(* IEC 61131-3 sources: cc_kush_rewrite/POUs/Bunker/POU/Hardware, 4 files *)

(* ---- FB_BunkerMotorErrors.st ---- *)
FUNCTION_BLOCK FB_BunkerMotorErrors
VAR_INPUT
	Bunker : REFERENCE TO ST_Bunker;
	xReset : BOOL; // Команда сброса зафиксированных ошибок
END_VAR
VAR_OUTPUT
	// Ошибки вибропитателей (индивидуально)
	xErrorVibFeeder1 : BOOL;
	xErrorVibFeeder2 : BOOL;
	xErrorMotorVibFeeder_Any : BOOL; // Ошибка хотя бы одного вибропитателя

	// Ошибки вибраторов (индивидуально)
	xErrorVibrator1 : BOOL;
	xErrorVibrator2 : BOOL;
	xErrorVibrator3 : BOOL;
	xErrorVibrator4 : BOOL;
	xErrorMotorVibrator_Any : BOOL; // Ошибка хотя бы одного вибратора

	// Ошибки бункера
	xErrorBunker : BOOL; // Ошибка бункера (люк, вес)

	// Состояние автоматических выключателей (QF)
	xQF_OkVibFeeder1 : BOOL;
	xQF_OkVibFeeder2 : BOOL;
	xQF_OkVibFeeder_All : BOOL;

	xQF_OkVibrator1 : BOOL;
	xQF_OkVibrator2 : BOOL;
	xQF_OkVibrator3 : BOOL;
	xQF_OkVibrator4 : BOOL;
	xQF_OkVibrator_All : BOOL;

	xQF_Ok_All : BOOL; // Все QF включены

	// Готовность VFD
	xVFD_ReadyVibFeeder1 : BOOL;
	xVFD_ReadyVibFeeder2 : BOOL;
	xVFD_ReadyVibFeeder_All : BOOL;

	xVFD_ReadyVibrator1 : BOOL;
	xVFD_ReadyVibrator2 : BOOL;
	xVFD_ReadyVibrator3 : BOOL;
	xVFD_ReadyVibrator4 : BOOL;
	xVFD_ReadyVibrator_All : BOOL;

	xVFD_Ready_All : BOOL; // Все VFD готовы
END_VAR
VAR
	// Внутренние переменные для текущих состояний ошибок (без фиксации)
	_xCurrentErrorVibFeeder1 : BOOL;
	_xCurrentErrorVibFeeder2 : BOOL;
	_xCurrentErrorVibrator1 : BOOL;
	_xCurrentErrorVibrator2 : BOOL;
	_xCurrentErrorVibrator3 : BOOL;
	_xCurrentErrorVibrator4 : BOOL;
	_xCurrentErrorBunker : BOOL;

	// RS-триггеры для фиксации ошибок
	_fbLatchErrorVibFeeder1 : RS;
	_fbLatchErrorVibFeeder2 : RS;
	_fbLatchErrorVibrator1 : RS;
	_fbLatchErrorVibrator2 : RS;
	_fbLatchErrorVibrator3 : RS;
	_fbLatchErrorVibrator4 : RS;
	_fbLatchErrorBunker : RS;
END_VAR

// ========================================
// FB_BunkerMotorErrors - Проверка ошибок моторов бункера
// ========================================
//
// НАЗНАЧЕНИЕ:
// - Проверка всех моторов бункера на ошибки
// - Фиксация ошибок через RS-триггеры (память до сброса)
// - Формирование индивидуальных флагов ошибок
// - Агрегирование ошибок
//
// МОТОРЫ:
// - MotorVibFeeder[1..2]: Вибропитатели (7.5 кВт)
// - MotorVibrator[1..4]: Вибраторы (0.62 кВт)
//
// ПРОВЕРЯЕМЫЕ ОШИБКИ:
// - Ошибка VFD (fbStateFailure: NC контакт - 0 = ошибка, 1 = норма)
// - Локальная ошибка VFD (xStateFailureLocal: программная установка ошибки)
//
// ЛОГИКА ФИКСАЦИИ:
// - При возникновении ошибки она фиксируется (SET в RS-триггер)
// - Ошибка сохраняется даже после устранения неисправности
// - Сброс всех зафиксированных ошибок через вход xReset
//
// ========================================

// ========================================
// ПРОВЕРКА ОШИБОК ВИБРОПИТАТЕЛЕЙ
// ========================================

// Вибропитатель 1
// fbStateFailure - NC контакт: 0 = ошибка VFD, 1 = норма
// Используем инвертированный сигнал (qxInvertedSignal: TRUE = ошибка)
_xCurrentErrorVibFeeder1 := Bunker.MotorVibFeeder[1].VFD.fbStateFailure.qxInvertedSignal
                         OR Bunker.MotorVibFeeder[1].VFD.xStateFailureLocal;

// Вибропитатель 2
_xCurrentErrorVibFeeder2 := Bunker.MotorVibFeeder[2].VFD.fbStateFailure.qxInvertedSignal
                         OR Bunker.MotorVibFeeder[2].VFD.xStateFailureLocal;

// Фиксируем ошибки через RS-триггеры
_fbLatchErrorVibFeeder1(SET := _xCurrentErrorVibFeeder1, RESET1 := xReset);
_fbLatchErrorVibFeeder2(SET := _xCurrentErrorVibFeeder2, RESET1 := xReset);

// Выходы - зафиксированные ошибки
xErrorVibFeeder1 := _fbLatchErrorVibFeeder1.Q1;
xErrorVibFeeder2 := _fbLatchErrorVibFeeder2.Q1;

xErrorMotorVibFeeder_Any := xErrorVibFeeder1 OR xErrorVibFeeder2;

// ========================================
// ПРОВЕРКА ОШИБОК ВИБРАТОРОВ
// ========================================

// Вибратор 1
_xCurrentErrorVibrator1 := Bunker.MotorVibrator[1].VFD.fbStateFailure.qxInvertedSignal
                        OR Bunker.MotorVibrator[1].VFD.xStateFailureLocal;

// Вибратор 2
_xCurrentErrorVibrator2 := Bunker.MotorVibrator[2].VFD.fbStateFailure.qxInvertedSignal
                        OR Bunker.MotorVibrator[2].VFD.xStateFailureLocal;

// Вибратор 3
_xCurrentErrorVibrator3 := Bunker.MotorVibrator[3].VFD.fbStateFailure.qxInvertedSignal
                        OR Bunker.MotorVibrator[3].VFD.xStateFailureLocal;

// Вибратор 4
_xCurrentErrorVibrator4 := Bunker.MotorVibrator[4].VFD.fbStateFailure.qxInvertedSignal
                        OR Bunker.MotorVibrator[4].VFD.xStateFailureLocal;

// Фиксируем ошибки через RS-триггеры
_fbLatchErrorVibrator1(SET := _xCurrentErrorVibrator1, RESET1 := xReset);
_fbLatchErrorVibrator2(SET := _xCurrentErrorVibrator2, RESET1 := xReset);
_fbLatchErrorVibrator3(SET := _xCurrentErrorVibrator3, RESET1 := xReset);
_fbLatchErrorVibrator4(SET := _xCurrentErrorVibrator4, RESET1 := xReset);

// Выходы - зафиксированные ошибки
xErrorVibrator1 := _fbLatchErrorVibrator1.Q1;
xErrorVibrator2 := _fbLatchErrorVibrator2.Q1;
xErrorVibrator3 := _fbLatchErrorVibrator3.Q1;
xErrorVibrator4 := _fbLatchErrorVibrator4.Q1;

xErrorMotorVibrator_Any := xErrorVibrator1 OR xErrorVibrator2 OR xErrorVibrator3 OR xErrorVibrator4;

// ========================================
// ПРОВЕРКА ОШИБОК БУНКЕРА
// ========================================

// Проверка положения люка (1 = закрыт, 0 = открыт)
// Открытый люк = ошибка
_xCurrentErrorBunker := NOT Bunker.fbStateHatch.qxSignal;

// Фиксируем ошибку через RS-триггер
_fbLatchErrorBunker(SET := _xCurrentErrorBunker, RESET1 := xReset);

// Выход - зафиксированная ошибка
xErrorBunker := _fbLatchErrorBunker.Q1;

// ========================================
// ПРОВЕРКА ГОТОВНОСТИ VFD
// ========================================
// fbStateRdyToStart - NO контакт: 1 = готов к пуску, 0 = не готов
// Готовность проверяется в реальном времени (без фиксации)

// Готовность VFD вибропитателей
xVFD_ReadyVibFeeder1 := Bunker.MotorVibFeeder[1].VFD.fbStateRdyToStart.qxSignal;
xVFD_ReadyVibFeeder2 := Bunker.MotorVibFeeder[2].VFD.fbStateRdyToStart.qxSignal;
xVFD_ReadyVibFeeder_All := xVFD_ReadyVibFeeder1 AND xVFD_ReadyVibFeeder2;

// Готовность VFD вибраторов
xVFD_ReadyVibrator1 := Bunker.MotorVibrator[1].VFD.fbStateRdyToStart.qxSignal;
xVFD_ReadyVibrator2 := Bunker.MotorVibrator[2].VFD.fbStateRdyToStart.qxSignal;
xVFD_ReadyVibrator3 := Bunker.MotorVibrator[3].VFD.fbStateRdyToStart.qxSignal;
xVFD_ReadyVibrator4 := Bunker.MotorVibrator[4].VFD.fbStateRdyToStart.qxSignal;
xVFD_ReadyVibrator_All := xVFD_ReadyVibrator1 AND xVFD_ReadyVibrator2 AND xVFD_ReadyVibrator3 AND xVFD_ReadyVibrator4;

// Общая готовность всех VFD
xVFD_Ready_All := xVFD_ReadyVibFeeder_All AND xVFD_ReadyVibrator_All;

// ========================================
// ПРОВЕРКА СОСТОЯНИЯ АВТОМАТИЧЕСКИХ ВЫКЛЮЧАТЕЛЕЙ (QF)
// ========================================
// fbStateQF - NO контакт: 1 = QF включен, 0 = QF выключен
// Состояние проверяется в реальном времени (без фиксации)
// Выключенный QF - не ошибка, но запуск мотора невозможен

// Состояние QF вибропитателей
xQF_OkVibFeeder1 := Bunker.MotorVibFeeder[1].fbStateQF.qxSignal;
xQF_OkVibFeeder2 := Bunker.MotorVibFeeder[2].fbStateQF.qxSignal;
xQF_OkVibFeeder_All := xQF_OkVibFeeder1 AND xQF_OkVibFeeder2;

// Состояние QF вибраторов
xQF_OkVibrator1 := Bunker.MotorVibrator[1].fbStateQF.qxSignal;
xQF_OkVibrator2 := Bunker.MotorVibrator[2].fbStateQF.qxSignal;
xQF_OkVibrator3 := Bunker.MotorVibrator[3].fbStateQF.qxSignal;
xQF_OkVibrator4 := Bunker.MotorVibrator[4].fbStateQF.qxSignal;
xQF_OkVibrator_All := xQF_OkVibrator1 AND xQF_OkVibrator2 AND xQF_OkVibrator3 AND xQF_OkVibrator4;

// Общее состояние всех QF
xQF_Ok_All := xQF_OkVibFeeder_All AND xQF_OkVibrator_All;

END_FUNCTION_BLOCK

(* ---- FB_BunkerSensors.st ---- *)
FUNCTION_BLOCK FB_BunkerSensors
VAR_INPUT
	Bunker : REFERENCE TO ST_Bunker;
	xReset : BOOL;
END_VAR
VAR_OUTPUT
	xErrorHatch : BOOL;     // Ошибка положения люка
END_VAR

// ========================================
// FB_BunkerSensors - Обработка датчиков безопасности бункера
// ========================================
//
// НАЗНАЧЕНИЕ:
// - Обработка датчиков безопасности (люк)
// - Аналог FB_DumperSensors / FB_ConveyorSensors
// - Предоставляет единую точку для проверки датчиков
//
// ВХОДЫ:
// - Bunker: ссылка на структуру бункера
// - xReset: команда сброса ошибок
//
// ВЫХОДЫ:
// - xErrorHatch: ошибка положения люка
//
// ========================================

// ========================================
// ПРОВЕРКА ПОЛОЖЕНИЯ ЛЮКА
// ========================================

// Проверка положения люка (1 = закрыт, 0 = открыт)
// Если люк открыт - ошибка
xErrorHatch := NOT Bunker.fbStateHatch.qxSignal;

// ПРИМЕЧАНИЕ: В будущем здесь могут быть добавлены другие датчики безопасности

END_FUNCTION_BLOCK

(* ---- FB_BunkerVibFeederMotors.st ---- *)
FUNCTION_BLOCK FB_BunkerVibFeederMotors
VAR_INPUT
	Bunker : REFERENCE TO ST_Bunker;
	xStart : BOOL;              // Команда запуска
	xStop : BOOL;               // Команда остановки
	xEmergencyStop : BOOL;      // Аварийная остановка
	xReset : BOOL;              // Сброс ошибок
	rTargetFrequency : REAL;    // Целевая частота (Гц)
END_VAR
VAR_OUTPUT
	eStage : E_StageActuator;   // IDLE/STARTING/WORK/STOPPING/FAULT
	rCurrentFrequency : REAL;   // Средняя частота двух моторов
	xStartingTimeout : BOOL;    // Флаг тайм-аута запуска
	xStoppingTimeout : BOOL;    // Флаг тайм-аута остановки
END_VAR
VAR
	STAGE : E_StageActuator := E_StageActuator.IDLE;

	// Таймеры контроля времени запуска/остановки
	tonTimerStarting : TON;     // Контроль времени запуска (STARTING → WORK)
	tonTimerStopping : TON;     // Контроль времени остановки (STOPPING → IDLE)
END_VAR

// ========================================
// FB_BunkerVibFeederMotors - Управление моторами вибропитателей бункера
// ========================================
//
// НАЗНАЧЕНИЕ:
// - Управление двумя вибропитателями (7.5 кВт каждый)
// - Прямой пуск/остановка (без плавного разгона)
// - Не знает про ППЗ и верхнеуровневую логику
// - Просто выполняет команды START/STOP
//
// ВХОДЫ:
// - xStart: команда запуска моторов
// - xStop: команда остановки моторов
// - xEmergencyStop: аварийная остановка
// - xReset: сброс аварии
// - rTargetFrequency: целевая частота (Гц)
//
// ВЫХОДЫ:
// - eStage: текущая стадия (IDLE/STARTING/WORK/STOPPING/FAULT)
// - rCurrentFrequency: текущая частота моторов (среднее)
// - xStartingTimeout: флаг тайм-аута запуска
// - xStoppingTimeout: флаг тайм-аута остановки
//
// ========================================

// ========================================
// ПРИОРИТЕТНАЯ ОБРАБОТКА АВАРИЙНОЙ ОСТАНОВКИ
// ========================================

IF xEmergencyStop THEN
	// Аварийная остановка: немедленное выключение VFD
	Bunker.MotorVibFeeder[1].VFD.qxStart := FALSE;
	Bunker.MotorVibFeeder[2].VFD.qxStart := FALSE;

	// Переход в FAULT
	STAGE := E_StageActuator.FAULT;
	tonTimerStarting(IN := FALSE);
	tonTimerStopping(IN := FALSE);
END_IF

// ========================================
// ПРОВЕРКА ТАЙМ-АУТОВ ВЫПОЛНЕНИЯ КОМАНД
// ========================================

// Тайм-аут запуска: если слишком долго в STARTING → аварийная остановка
tonTimerStarting(
	IN := (STAGE = E_StageActuator.STARTING),
	PT := TIME_TIMEOUT_START_BUNKER
);

IF tonTimerStarting.Q THEN
	xStartingTimeout := TRUE;
	// Аварийная остановка: немедленное выключение VFD
	Bunker.MotorVibFeeder[1].VFD.qxStart := FALSE;
	Bunker.MotorVibFeeder[2].VFD.qxStart := FALSE;
	// Переход в FAULT
	STAGE := E_StageActuator.FAULT;
	tonTimerStarting(IN := FALSE);
END_IF

// Тайм-аут остановки: если слишком долго в STOPPING → аварийная остановка
tonTimerStopping(
	IN := (STAGE = E_StageActuator.STOPPING),
	PT := TIME_TIMEOUT_STOP_BUNKER
);

IF tonTimerStopping.Q THEN
	xStoppingTimeout := TRUE;
	// Аварийная остановка: немедленное выключение VFD
	Bunker.MotorVibFeeder[1].VFD.qxStart := FALSE;
	Bunker.MotorVibFeeder[2].VFD.qxStart := FALSE;
	// Переход в FAULT
	STAGE := E_StageActuator.FAULT;
	tonTimerStopping(IN := FALSE);
END_IF

// ========================================
// АВТОМАТ УПРАВЛЕНИЯ МОТОРАМИ
// ========================================

CASE STAGE OF
	E_StageActuator.IDLE:
		// Сброс команд
		Bunker.MotorVibFeeder[1].VFD.qxStart := FALSE;
		Bunker.MotorVibFeeder[2].VFD.qxStart := FALSE;

		// Команда запуска
		IF xStart AND NOT xEmergencyStop THEN
			STAGE := E_StageActuator.STARTING;
		END_IF

	E_StageActuator.STARTING:
		// Проверка команды остановки во время запуска
		IF xStop THEN
			// Прервать запуск и перейти к остановке
			STAGE := E_StageActuator.STOPPING;
		END_IF

		// Команда ПУСК на VFD
		Bunker.MotorVibFeeder[1].VFD.qxStart := TRUE;
		Bunker.MotorVibFeeder[2].VFD.qxStart := TRUE;

		// Проверка обратной связи VFD
		IF Bunker.MotorVibFeeder[1].VFD.fbStateIsWorking.qxSignal
		   AND Bunker.MotorVibFeeder[2].VFD.fbStateIsWorking.qxSignal
		THEN
			// Сброс таймера запуска (успешный запуск)
			tonTimerStarting(IN := FALSE);
			STAGE := E_StageActuator.WORK;
		END_IF

	E_StageActuator.WORK:
		// Нормальная работа
		// Команда остановки - переход в STOPPING
		IF xStop THEN
			STAGE := E_StageActuator.STOPPING;
		END_IF

	E_StageActuator.STOPPING:
		// Остановка VFD
		Bunker.MotorVibFeeder[1].VFD.qxStart := FALSE;
		Bunker.MotorVibFeeder[2].VFD.qxStart := FALSE;

		// Проверка остановки VFD (обратная связь)
		IF NOT Bunker.MotorVibFeeder[1].VFD.fbStateIsWorking.qxSignal
		   AND NOT Bunker.MotorVibFeeder[2].VFD.fbStateIsWorking.qxSignal
		THEN
			// Сброс таймера остановки (успешная остановка)
			tonTimerStopping(IN := FALSE);
			STAGE := E_StageActuator.IDLE;
		END_IF

	E_StageActuator.FAULT:
		// Состояние аварии - ожидание сброса
		// Выход из FAULT по команде xReset
		IF xReset THEN
			STAGE := E_StageActuator.IDLE;
			xStartingTimeout := FALSE; // Сброс флага тайм-аута запуска
			xStoppingTimeout := FALSE; // Сброс флага тайм-аута остановки
		END_IF
END_CASE;

// ========================================
// ЗАДАНИЕ ЧАСТОТЫ МОТОРОВ
// ========================================

// Установка частоты напрямую (без плавного разгона)
// В режимах STARTING и WORK частота = rTargetFrequency
// В остальных режимах (IDLE, STOPPING, FAULT) частота = 0
IF STAGE = E_StageActuator.STARTING OR STAGE = E_StageActuator.WORK THEN
	Bunker.MotorVibFeeder[1].VFD.qrOutFrequency := rTargetFrequency;
	Bunker.MotorVibFeeder[2].VFD.qrOutFrequency := rTargetFrequency;
ELSE
	Bunker.MotorVibFeeder[1].VFD.qrOutFrequency := 0.0;
	Bunker.MotorVibFeeder[2].VFD.qrOutFrequency := 0.0;
END_IF;

// ========================================
// ВЫХОДЫ
// ========================================

// Текущая стадия
eStage := STAGE;

// Текущая частота (среднее значение двух моторов)
rCurrentFrequency := (Bunker.MotorVibFeeder[1].VFD.rActualFrequency
                    + Bunker.MotorVibFeeder[2].VFD.rActualFrequency) / 2.0;

END_FUNCTION_BLOCK

(* ---- FB_BunkerVibratorMotors.st ---- *)
FUNCTION_BLOCK FB_BunkerVibratorMotors
VAR_INPUT
	Bunker : REFERENCE TO ST_Bunker;
	xEmergencyStop : BOOL;              // Аварийная остановка
	xReset : BOOL;                      // Сброс ошибок
	eVibratorMode : E_StateRemote;      // Auto/Manual/Repair
	xManualStart : BOOL;                // СТАРТ в ручном режиме
	xManualStop : BOOL;                 // СТОП в ручном режиме
	xSelectedVibrators : ARRAY[1..4] OF BOOL;  // Выбор вибраторов (галочки)
	rTargetFrequency : REAL;            // Целевая частота
	stVibratorSettings : ST_BunkerVibratorSettings; // Параметры цикла
	xEnableAutoMode : BOOL;             // Разрешение автоматического режима (только в WORK вибропитателей)
END_VAR
VAR_OUTPUT
	eStage : E_StageActuator;           // IDLE/STARTING/WORK/STOPPING/FAULT
	xVibratorAutoActive : BOOL;         // Флаг активной работы (Auto)
	xVibratorManualRunActive : BOOL;    // Флаг активной работы (Manual)
END_VAR
VAR
	STAGE : E_StageActuator := E_StageActuator.IDLE;  // Текущая стадия
	tonVibratorActive : TON;            // Таймер активной работы (Auto)
	tonVibratorPause : TON;             // Таймер паузы (Auto)
	i : INT;

	// Переменные для последовательного запуска вибраторов
	tonSequentialStart : TON;           // Таймер шага последовательного запуска
	nSequentialIndex : INT := 0;        // Текущий индекс в последовательности запуска (0 = не запущен, 1-4 = номер вибратора)
	axVibratorStarted : ARRAY[1..4] OF BOOL; // Флаги запущенных вибраторов в текущем цикле ACTIVE
	xSequentialStartComplete : BOOL;    // Все выбранные вибраторы запущены
END_VAR

// ========================================
// FB_BunkerVibratorMotors - Управление вибраторами бункера
// ========================================
//
// НАЗНАЧЕНИЕ:
// - Управление 4 вибраторами (0.62 кВт каждый)
// - 3 режима: Auto (цикл), Manual (выборочное управление), Repair (остановка)
// - Auto режим: ACTIVE (работа) ↔ PAUSE (пауза) циклически
// - Manual режим: индивидуальный выбор через галочки + СТАРТ/СТОП
// - Не знает про вибропитатели и верхнеуровневую логику
//
// ВХОДЫ:
// - xEmergencyStop: аварийная остановка
// - xReset: сброс ошибок
// - eVibratorMode: режим управления (Auto/Manual/Repair)
// - xManualStart: команда СТАРТ в ручном режиме
// - xManualStop: команда СТОП в ручном режиме
// - xSelectedVibrators[1..4]: выбор вибраторов (галочки)
// - rTargetFrequency: целевая частота (Гц)
// - stVibratorSettings: параметры цикла (TIME_ACTIVE, TIME_PAUSE_VIBRATOR и т.д.)
// - xEnableAutoMode: разрешение автоматического режима (TRUE только в WORK вибропитателей)
//
// ВЫХОДЫ:
// - eStage: текущая стадия (IDLE/STARTING/WORK/STOPPING/FAULT)
// - xVibratorAutoActive: флаг активной работы в авто режиме
// - xVibratorManualRunActive: флаг активной работы в ручном режиме
//
// ========================================

// ========================================
// ПРИОРИТЕТНАЯ ОБРАБОТКА АВАРИЙНОЙ ОСТАНОВКИ
// ========================================

IF xEmergencyStop THEN
	// Остановка всех VFD вибраторов
	Bunker.MotorVibrator[1].VFD.qxStart := FALSE;
	Bunker.MotorVibrator[2].VFD.qxStart := FALSE;
	Bunker.MotorVibrator[3].VFD.qxStart := FALSE;
	Bunker.MotorVibrator[4].VFD.qxStart := FALSE;

	// Сброс таймеров и флагов
	tonVibratorActive(IN := FALSE);
	tonVibratorPause(IN := FALSE);
	tonSequentialStart(IN := FALSE);
	xVibratorManualRunActive := FALSE;
	xVibratorAutoActive := FALSE;
	nSequentialIndex := 0;
	xSequentialStartComplete := FALSE;
	FOR i := 1 TO 4 BY 1 DO
		axVibratorStarted[i] := FALSE;
	END_FOR;

	// Переход в FAULT
	STAGE := E_StageActuator.FAULT;
END_IF

// ========================================
// НОРМАЛЬНАЯ РАБОТА ВИБРАТОРОВ
// ========================================

IF NOT xEmergencyStop THEN
	CASE eVibratorMode OF
		// ========================================
		// РЕЖИМ АВТОМАТИЧЕСКИЙ - циклическая работа по таймеру
		// ========================================
		E_StateRemote.Auto:
			// Автоматический режим работает только при разрешении (в WORK вибропитателей)
			IF xEnableAutoMode THEN
				// Установка частоты для вибраторов в автоматическом режиме
				FOR i := 1 TO AMOUNT_BUNKER_MOTOR_VIBRATOR BY 1 DO
					Bunker.MotorVibrator[i].VFD.qrOutFrequency := rTargetFrequency;
				END_FOR;

				// Таймеры автоматического цикла
				tonVibratorActive(PT := stVibratorSettings.TIME_ACTIVE);
				tonVibratorPause(PT := stVibratorSettings.TIME_PAUSE_VIBRATOR);
				tonSequentialStart(PT := TIME_VIBRATOR_SEQUENTIAL_START_STEP);

				// Логика автоматического цикла (ACTIVE ↔ PAUSE)
				IF NOT xVibratorAutoActive THEN
					// Состояние PAUSE - ждем окончания паузы
					IF tonVibratorPause.Q THEN
						// Пауза завершена - переход в ACTIVE
						tonVibratorPause(IN := FALSE);
						xVibratorAutoActive := TRUE;

						// Сброс состояния последовательного запуска
						nSequentialIndex := 0;
						xSequentialStartComplete := FALSE;
						FOR i := 1 TO 4 BY 1 DO
							axVibratorStarted[i] := FALSE;
						END_FOR;
						tonSequentialStart(IN := FALSE);
						tonVibratorActive(IN := FALSE); // Таймер ACTIVE запустится после завершения последовательного запуска

						// Переход в WORK (вибраторы будут запускаться последовательно)
						STAGE := E_StageActuator.WORK;
					ELSIF NOT tonVibratorPause.IN THEN
						// Первый запуск - сразу в ACTIVE
						xVibratorAutoActive := TRUE;

						// Сброс состояния последовательного запуска
						nSequentialIndex := 0;
						xSequentialStartComplete := FALSE;
						FOR i := 1 TO 4 BY 1 DO
							axVibratorStarted[i] := FALSE;
						END_FOR;
						tonSequentialStart(IN := FALSE);
						tonVibratorActive(IN := FALSE); // Таймер ACTIVE запустится после завершения последовательного запуска

						// Переход в WORK (вибраторы будут запускаться последовательно)
						STAGE := E_StageActuator.WORK;
					ELSE
						// Пауза активна - IDLE
						STAGE := E_StageActuator.IDLE;
					END_IF;
				ELSE
					// Состояние ACTIVE - последовательный запуск вибраторов

					// Логика последовательного запуска (если ещё не все запущены)
					IF NOT xSequentialStartComplete THEN
						// Проверка таймера для запуска следующего вибратора
						IF NOT tonSequentialStart.IN OR tonSequentialStart.Q THEN
							// Сброс таймера и поиск следующего выбранного вибратора
							tonSequentialStart(IN := FALSE);

							// Ищем следующий выбранный вибратор, который ещё не запущен
							FOR i := 1 TO 4 BY 1 DO
								IF xSelectedVibrators[i] AND NOT axVibratorStarted[i] THEN
									// Найден следующий вибратор для запуска
									Bunker.MotorVibrator[i].VFD.qxStart := TRUE;
									axVibratorStarted[i] := TRUE;
									nSequentialIndex := i;
									tonSequentialStart(IN := TRUE); // Запуск таймера для следующего
									EXIT; // Выход из цикла - запускаем только один за раз
								END_IF;
							END_FOR;

							// Проверка: все ли выбранные вибраторы запущены
							xSequentialStartComplete := TRUE;
							FOR i := 1 TO 4 BY 1 DO
								IF xSelectedVibrators[i] AND NOT axVibratorStarted[i] THEN
									xSequentialStartComplete := FALSE;
									EXIT;
								END_IF;
							END_FOR;

							// Если все запущены - остановить таймер последовательного запуска и запустить таймер ACTIVE
							IF xSequentialStartComplete THEN
								tonSequentialStart(IN := FALSE);
								tonVibratorActive(IN := TRUE); // Таймер ACTIVE начинается после запуска всех выбранных вибраторов
							END_IF;
						END_IF;
					END_IF;

					// Проверка окончания активной работы (только если все вибраторы уже запущены)
					IF xSequentialStartComplete AND tonVibratorActive.Q THEN
						// Активная работа завершена - переход в PAUSE
						tonVibratorActive(IN := FALSE);
						tonVibratorPause(IN := TRUE);
						tonSequentialStart(IN := FALSE);
						xVibratorAutoActive := FALSE;
						xSequentialStartComplete := FALSE;
						nSequentialIndex := 0;

						// Остановка всех вибраторов
						FOR i := 1 TO 4 BY 1 DO
							Bunker.MotorVibrator[i].VFD.qxStart := FALSE;
							axVibratorStarted[i] := FALSE;
						END_FOR;

						// Переход в IDLE (пауза)
						STAGE := E_StageActuator.IDLE;
					ELSE
						// Активная работа - WORK
						STAGE := E_StageActuator.WORK;
					END_IF;
				END_IF;
			ELSE
				// Вне WORK вибропитателей - остановка автоматического цикла
				tonVibratorActive(IN := FALSE);
				tonVibratorPause(IN := FALSE);
				tonSequentialStart(IN := FALSE);
				xVibratorAutoActive := FALSE;
				xSequentialStartComplete := FALSE;
				nSequentialIndex := 0;

				// Остановка всех вибраторов
				FOR i := 1 TO 4 BY 1 DO
					Bunker.MotorVibrator[i].VFD.qxStart := FALSE;
					axVibratorStarted[i] := FALSE;
				END_FOR;

				// Переход в IDLE
				STAGE := E_StageActuator.IDLE;
			END_IF;

		// ========================================
		// РЕЖИМ РУЧНОЙ - индивидуальное управление через выбор + старт/стоп
		// ========================================
		E_StateRemote.Manual:
			// Команда СТАРТ активирует флаг запуска
			IF xManualStart THEN
				xVibratorManualRunActive := TRUE;
			END_IF

			// Команда СТОП останавливает ВСЕ вибраторы и сбрасывает флаг
			IF xManualStop THEN
				xVibratorManualRunActive := FALSE;
				Bunker.MotorVibrator[1].VFD.qxStart := FALSE;
				Bunker.MotorVibrator[2].VFD.qxStart := FALSE;
				Bunker.MotorVibrator[3].VFD.qxStart := FALSE;
				Bunker.MotorVibrator[4].VFD.qxStart := FALSE;
			END_IF

			// Если флаг запуска активен - управляем вибраторами через галочки выбора
			IF xVibratorManualRunActive THEN
				// Каждый вибратор работает только если он выбран (галочка установлена)
				Bunker.MotorVibrator[1].VFD.qxStart := xSelectedVibrators[1];
				Bunker.MotorVibrator[2].VFD.qxStart := xSelectedVibrators[2];
				Bunker.MotorVibrator[3].VFD.qxStart := xSelectedVibrators[3];
				Bunker.MotorVibrator[4].VFD.qxStart := xSelectedVibrators[4];

				// Проверка: хотя бы один вибратор выбран → WORK
				IF xSelectedVibrators[1] OR xSelectedVibrators[2] OR xSelectedVibrators[3] OR xSelectedVibrators[4] THEN
					STAGE := E_StageActuator.WORK;
				ELSE
					STAGE := E_StageActuator.IDLE;
				END_IF;
			ELSE
				// Флаг запуска неактивен - IDLE
				STAGE := E_StageActuator.IDLE;
			END_IF

			// Установка частоты для вибраторов в ручном режиме
			FOR i := 1 TO AMOUNT_BUNKER_MOTOR_VIBRATOR BY 1 DO
				Bunker.MotorVibrator[i].VFD.qrOutFrequency := rTargetFrequency;
			END_FOR;

		// ========================================
		// РЕЖИМ РЕМОНТ - все вибраторы остановлены
		// ========================================
		E_StateRemote.Repair:
			xVibratorManualRunActive := FALSE;
			xVibratorAutoActive := FALSE;
			Bunker.MotorVibrator[1].VFD.qxStart := FALSE;
			Bunker.MotorVibrator[2].VFD.qxStart := FALSE;
			Bunker.MotorVibrator[3].VFD.qxStart := FALSE;
			Bunker.MotorVibrator[4].VFD.qxStart := FALSE;

			// Режим ремонт - IDLE
			STAGE := E_StageActuator.IDLE;
	END_CASE
END_IF; // Конец IF NOT xEmergencyStop

// ========================================
// ВЫХОД ИЗ FAULT ПО КОМАНДЕ СБРОСА
// ========================================

IF STAGE = E_StageActuator.FAULT AND xReset THEN
	STAGE := E_StageActuator.IDLE;
END_IF

// ========================================
// ВЫХОДЫ
// ========================================

eStage := STAGE;

END_FUNCTION_BLOCK
